FUNCTION_BLOCK EL1819
VAR
	_io : EL1xx9_Data;
	{attribute addProperty Name "WcState"}
	_wcState : WcStateInputToggle;
	{attribute addProperty Name "Info data"}
	_infoData : InfoDataBase;
END_VAR

PROPERTY IO : REFERENCE TO EL1xx9_Data
GET
IO REF= _io;
END_GET
END_PROPERTY

PROPERTY WcState : REFERENCE TO WcStateInputToggle
GET
WcState REF= _wcState;
END_GET
END_PROPERTY

END_FUNCTION_BLOCK

(* stored: Version 1.1.0.1, ProductVersion 3.1.4024.9
   POU EL1819: Id {8008e8bb-794a-07da-3020-b6b84382aa1f}, SpecialFunc None
   Property IO: Id {ec765bba-0363-0d3c-1bfe-ef71bcc1255c}
   Get Get: Id {db0167a7-3e4b-08f4-0c9c-debc2e69095b}
   Property WcState: Id {d3a75c52-7d7a-0094-247d-5c726d72ee84}
   Get Get: Id {88880b28-6dc7-0794-0584-23ea6560796c} *)
